{attribute 'qualified_only'}
{attribute 'qualified_only'}
VAR_GLOBAL
    // InCmd
    {attribute 'OPC.UA.DA' := '1'}
    {attribute 'OPC.UA.DA.StructuredType' := '1'}
    g_stBigBagChangeHandlerInCmd      : ST_BigBagChangeHandlerInCmd;

    // InValues
    {attribute 'OPC.UA.DA' := '1'}
    {attribute 'OPC.UA.DA.StructuredType' := '1'}
    g_stBigBagChangeHandlerInValues   : ST_BigBagChangeHandlerInValues;


    // Status
    {attribute 'OPC.UA.DA' := '1'}
    {attribute 'OPC.UA.DA.StructuredType' := '1'}
    g_stBigBagChangeHandlerStatus     : ST_BigBagChangeHandlerStatus;
	
	// OutValues
    {attribute 'OPC.UA.DA' := '1'}
    {attribute 'OPC.UA.DA.StructuredType' := '1'}
    g_stBigBagChangeHandlerOutValues   : ST_BigBagChangeHandlerOutValues;
	
END_VAR

(* stored: Version 1.1.0.1, ProductVersion 3.1.4024.16
   GVL GVL_BigBagChangeHandler: Id {9cace0c0-b90d-459b-9382-79cea52ba527} *)
